# EPICS substitutions: iocBoot/ioc-xpp-gige-02/ioc-xpp-gige-02.substitutions
# IOC archive file
## Replace IOC:XPP:GIGE:02 with the PV prefix used for
## iocAdmin PV's on this IOC

# Generate IOC archive request
file archive_gige.archive
{
	{ IOC = "IOC:XPP:GIGE:02" }
}
